Fanuc KAREL source: kf00092.KL

PROGRAM KF00092
%STACKSIZE=65535
%PRIORITY=65535
%NOLOCKGROUP
VAR
I : INTEGER
J : INTEGER
X : REAL
Y : REAL
B : BOOLEAN
C : BOOLEAN
TXT : STRING[80]
TXT2 : STRING[80]
AI : ARRAY[4] OF INTEGER
BI : ARRAY[4] OF INTEGER
P : XYZWPR
JP : JOINTPOS9
PF : POSITION
STATUS : INTEGER
-- UNRESOLVED DECLARATIONS (source type spelling not recovered)
-- V1 : TYPE_0x0013 (type_u16=0x0013)
-- V2 : TYPE_0x0013 (type_u16=0x0013)
BEGIN
-- UNSAFE_SOURCE_IR line 21: field_offset(V1,0) = 1065353216
-- UNSAFE_SOURCE_IR line 22: field_offset(V2,4) = 1065353216
-- UNRESOLVED_PC line 23 opcodes [49 49 93 4A] marker_code=40
END KF00092
